Staubli VAL3: Pallet.dtx

bool bExit
bool bListRefresh
bool bUserRefresh
public frame fFrame = {fatherId=world[0]}
mdesc mNomSpeed
num nPage = 1
num nSelected
num nType
public pallet uPallet{}
  [pallet1]
    frame fFrame
    num ndX
    num ndY
    pointRx pO = {x=493.537278, y=141.157682, z=-16.022447, rx=-172.031241, ry=0.156426, rz=65.99326, shoulder=lefty, elbow=epositive, wrist=wpositive, fatherId=world[0]}
    pointRx pStart
    pointRx pX
    pointRx pY
    string sToolName = "tool6"
  [pallet2]
    frame fFrame
    num ndX
    num ndY
    pointRx pO = {x=493.537278, y=141.157682, z=-16.022447, rx=-172.031241, ry=0.156426, rz=65.99326, shoulder=lefty, elbow=epositive, wrist=wpositive, fatherId=world[0]}
    pointRx pStart
    pointRx pX
    pointRx pY
    string sToolName
pointRx pPonit[3]
  [0] = {x=493.537278, y=141.157682, z=-16.022447, rx=-172.031241, ry=0.156426, rz=65.99326, fatherId=world[0]}
  [1] = {fatherId=world[0]}
  [2] = {fatherId=world[0]}
string sFrameName
string sItem = "pallet1"
string sList[2]
  [0] = "pallet1"
  [1] = "pallet2"
string sListItemValue[7]
  [3] = "0    "
  [4] = "0    "
  [6] = "tool6"
string sParameter[7]
  [0] = "原点     :          "
  [1] = "X点      :          "
  [2] = "Y点      :          "
  [3] = "dX       :0         "
  [4] = "dY       :0         "
  [5] = "起点     :          "
  [6] = "工具     :tool6     "
tool tTool = {fatherId=flange[0], ioLink=valve1}
